//TODO: set methods to enable all following, pneumatic cylinder activation, error handling

FUNCTION_BLOCK FB_GantryHoldDown
VAR_INPUT
	robot				: FB_Robot; //robot_object
END_VAR
VAR_OUTPUT
END_VAR
VAR
	//MC_functions, called in methods
	fbMC_PowerWest		: MC_Power;
	fbMC_PowerEast		: MC_Power;
	fbMC_SyncEastWest	: MC_MoveAbsolute;
	fbMC_MoveAbsWest1	: MC_MoveAbsolute;
	fbMC_MoveAbsWest2	: MC_MoveAbsolute;
	fbMC_HomeWest		: MC_Home;
	fbMC_HomeEast		: MC_Home;
	fbMC_SyncAxes		: MC_GearIn;
	Aborting			: MC_BufferMode;
	
	//Inputs
	ls1NE AT %I* 		: BOOL;
	ls3NW AT %I* 		: BOOL;
	
	//Enable bools
	executeEnableWest	: BOOL;
	executeEnableEast	: BOOL;
	executeHomeWest		: BOOL;
	executeHomeEast		: BOOL;
	executeFollow		: BOOL;
	executeSync			: BOOL := TRUE;
	executeCylinders	: BOOL;
	
	followVariable		: BOOL:= TRUE; //Set for following robot
	
	//Pneumatic cylinders
	cylindersNorth 			AT %Q* : BOOL;
	cylindersCentreNorth	AT %Q* : BOOL;
	cylindersCentreSouth	AT %Q* : BOOL;
	cylindersSouth			AT %Q* : BOOL;

	pbTableWest				AT %I* : BOOL;
	pbTableEast				AT %I* : BOOL;
	
	pbTableWestLast: BOOL;
	pbTableEastLast: BOOL;
	pbTableWestLastTrig: R_TRIG;
	pbTableEastLastTriq: R_TRIG;
	cylinderTableWest		AT %Q* : BOOL := FALSE;
	cylinderTableEast		AT %Q* : BOOL := FALSE;
	
	//Variable to be set by program being run
	LEN_WOOD : LREAL := 2133; //mm, length of wood being clamped

END_VAR

GVL_Axes.AxisWest.ReadStatus();
GVL_Axes.AxisEast.ReadStatus();
Enable_Axes();
Home_Axes();
Couple_Axes();
Follow_Robot();
Cylinder_Set_Cutting();
Load_Tables();

METHOD Couple_Axes
VAR_INPUT
END_VAR
fbMC_SyncAxes(
	Master:= GVL_Axes.AxisWest, 
	Slave:= GVL_Axes.AxisEast, 
	Execute:= executeSync, 
	RatioNumerator:= 1);
END_METHOD

METHOD Cylinder_Set_Cutting
VAR_INPUT
END_VAR
VAR
	POS_CYLINDER_NORTH : LREAL := 76.5; //mm, position of north pneum cylinder relative to gantry plate
	POS_CYLINDER_NORTHCENTRE : LREAL := 229.62; //mm, position of centre north pneum cylinder relative to gantry plate
	POS_CYLINDER_SOUTHCENTRE : LREAL := 712.212; //mm, position of centre south pneum cylinder relative to gantry plate
	POS_CYLINDER_SOUTH : LREAL := 867.832; //mm, position of south pneum cylinder relative to gantry plate
	POS_TABLE_NORTH : LREAL := 474.14; //mm, position of table start WRT Zero
	FACTOR_OF_SAFETY : LREAL := 100; //mm, distance from edge of table cylinders will rise
END_VAR
IF executeCylinders THEN
	IF GVL_Axes.AxisWest.NcToPlc.ActPos < POS_TABLE_NORTH + FACTOR_OF_SAFETY - POS_CYLINDER_NORTH THEN
		cylindersNorth := 1;
		IF GVL_Axes.AxisWest.NcToPlc.ActPos < POS_TABLE_NORTH + FACTOR_OF_SAFETY - POS_CYLINDER_NORTHCENTRE THEN
			cylindersCentreNorth := 1;
		ELSE
			cylindersCentreNorth := 0;
		END_IF
	ELSE
		cylindersNorth := 0;
	END_IF
	
	IF GVL_Axes.AxisWest.NcToPlc.ActPos > POS_TABLE_NORTH + LEN_WOOD - FACTOR_OF_SAFETY - POS_CYLINDER_SOUTH THEN
		cylindersSouth := 1;
		IF GVL_Axes.AxisWest.NcToPlc.ActPos > POS_TABLE_NORTH + LEN_WOOD - FACTOR_OF_SAFETY - POS_CYLINDER_SOUTHCENTRE THEN
			cylindersCentreSouth := 1;
		ELSE 
			cylindersCentreSouth := 0;
		END_IF
	ELSE
		cylindersSouth := 0;
	END_IF
END_IF
END_METHOD

METHOD Enable_Axes : BOOL
VAR_INPUT
END_VAR
//IF GVL_Axes.AxisWest.Status.Disabled THEN
//	executeEnableWest := TRUE;
//END_IF

//IF GVL_Axes.AxisEast.Status.Disabled THEN
//	executeEnableEast := TRUE;
//END_IF

fbMC_PowerWest(
		Axis:= GVL_Axes.AxisWest, 
		Enable:= executeEnableWest, 
		Enable_Positive:= executeEnableWest, 
		Enable_Negative:= executeEnableWest, 
		Override:= 100.0);
		
fbMC_PowerWest(
		Axis:= GVL_Axes.AxisEast, 
		Enable:= executeEnableEast, 
		Enable_Positive:= executeEnableEast, 
		Enable_Negative:= executeEnableEast, 
		Override:= 100.0);
END_METHOD

METHOD Follow_Robot
VAR_INPUT
END_VAR

VAR
	targetPosition: LREAL;
	accel: LREAL:=600;
	decel: LREAL:=600;
	jer:   LREAL:=1200;
	vel: LREAL:= 170;
END_VAR
//Set target position to middle of robot tool
targetPosition := (robot.y_pose - GVL_SERVO_ROBOT_CONST.MIN_POS_ROBOT) * GVL_SERVO_ROBOT_CONST.DIFFERENCE_SERVOWEST/GVL_SERVO_ROBOT_CONST.DIFFERENCE_ROBOT;
IF targetPosition < GVL_SERVO_ROBOT_CONST.MIN_POS_SERVOWEST THEN
	targetPosition := GVL_SERVO_ROBOT_CONST.MIN_POS_SERVOWEST;
ELSIF targetPosition > GVL_SERVO_ROBOT_CONST.MAX_POS_SERVOWEST THEN
	targetPosition := GVL_SERVO_ROBOT_CONST.MAX_POS_SERVOWEST;
END_IF

//If target position - current position > threshold, hold robot

followVariable := NOT followVariable;

IF executeFollow AND GVL_Axes.AxisWest.Status.Homed THEN
	fbMC_MoveAbsWest1(
		Axis:= GVL_Axes.AxisWest, 
		Execute:= followVariable, 
		Position:= targetPosition, 
		Velocity:= vel,
		Acceleration:= accel, 
		Deceleration:= decel,
		Jerk:= jer, 
		BufferMode:= Aborting);
	
	fbMC_MoveAbsWest2(
		Axis:= GVL_Axes.AxisWest, 
		Execute:= NOT followVariable, 
		Position:= targetPosition, 
		Velocity:= vel,
		Acceleration:= accel, 
		Deceleration:= decel,
		Jerk:= jer, 
		BufferMode:= Aborting);
END_IF
END_METHOD

METHOD Home_Axes
VAR_INPUT
END_VAR
	fbMC_HomeWest(
		Axis:= GVL_Axes.AxisWest, 
		Execute:= executeHomeWest, 
		Position:= GVL_SERVO_ROBOT_CONST.POSITION_LIMIT_SWITCH, 
		HomingMode:= MC_DefaultHoming, 
		bCalibrationCam:= NOT ls3NW);
	
//	fbMC_HomeEast(
//		Axis:= GVL_Axes.AxisEast, 
//		Execute:= executeHomeEast, 
//		Position:= 403, 
//		HomingMode:= MC_DefaultHoming, 
//		bCalibrationCam:= NOT ls1NE);
END_METHOD

METHOD Load_Tables
VAR_INPUT
END_VAR
IF pbTableWest AND NOT pbTableWestLast THEN
	cylinderTableWest := NOT cylinderTableWest;
END_IF

pbTableWestLast := pbTableWest;

IF pbTableEast AND NOT pbTableEastLast THEN
	cylinderTableEast := NOT cylinderTableEast;
END_IF

pbTableEastLast := pbTableEast;
END_METHOD

END_FUNCTION_BLOCK

(* stored: Version 1.1.0.1, ProductVersion 3.1.4024.12
   POU FB_GantryHoldDown: Id {212016f5-1181-4eaa-b089-a8c72c29c00d}, SpecialFunc None
   Method Couple_Axes: Id {5d338716-a070-49d0-a1b0-90505ad66513}
   Method Cylinder_Set_Cutting: Id {80c33305-3d27-491c-90ce-c1e0d842bbab}
   Method Enable_Axes: Id {c19824d3-7d09-4504-aec2-151759bbf50b}
   Method Follow_Robot: Id {56fb3307-d26a-436e-8a13-67eb97620809}
   Method Home_Axes: Id {47d775d5-845e-4f32-9b48-f325228313c3}
   Method Load_Tables: Id {7ee35345-9ea6-48dd-a062-6897bfc4de67} *)
